FUNCTION_BLOCK FB_MoveSS_Exte
VAR_INPUT
	enable	:BOOL;
	ref		:AXIS_REF;
	jogF	:BOOL;
	jogB	:BOOL;
	Acceleration		:LREAL;
	Deceleration		:LREAL;
	Jerk				:LREAL;
END_VAR
VAR_OUTPUT	
END_VAR
VAR
	MC_Read:MC_ReadStatus;
	MC_ABS:MC_MoveAbsolute;
	MC_REL:MC_MoveRelative;
	MC_Jog:MC_Jog;
	
	MC_ABS1:MC_MoveAbsolute;
	MC_ABS2:MC_MoveAbsolute;
	MC_VELO:MC_MoveVelocity;
	
	step1,step2,step3		:INT;	
	R_TRIG1,R_TRIG2,R_TRIG3	:R_TRIG;
	R_TRIG_done				:R_TRIG;
	ton_NotMoving			:TON;
	ton_Moving				:TON;
	rel_do					:BOOL;
	abs_do					:BOOL;
	jogF_do					:BOOL;
	jogB_do					:BOOL;
	
	abs_do1,abs_do2,velo_do	:BOOL;
	error					:BOOL;

	MoveAbsolute_Busy		:BOOL;
	MoveConstantVelocity_Busy:BOOL;
	MoveRelative_Busy		:BOOL;
	jog_EN					:BOOL;
	FB_START_r_trig:		R_TRIG;
	start					:BOOL;
	jog_f_trig				:F_TRIG;
	ton_NotMoving_r_trig:Tc2_Standard.R_TRIG;
END_VAR
VAR_IN_OUT 
	MoveRelExe					:BOOL;
	MoveAbsExe					:BOOL;
	MoveConstantVelocityExe		:BOOL;//
	Velo						:LREAL;	//mm/s
	TargetRel					:LREAL;//mm
	TargetAbs					:LREAL;//mm
	constantvelocityStart		:LREAL;//mm		The position to start moving with a constant velocity
												//      0 < ConstantVelocityStart< ConstanVelocityEnd< RequestedPosition
	constanvelocityEnd			:LREAL;//mm		The position to end moving with a constant velocity											
	Done						:BOOL;
	NotMovingTimeOut 			:BOOL;
	SpeedNotReach				:BOOL;
END_VAR

(*********************NOT MOVING TIMEOUT***************************)
FB_START_r_trig(CLK:=jogF OR jogB OR MoveRelExe OR MoveAbsExe OR MoveConstantVelocityExe  , Q=> );
IF FB_START_r_trig.Q THEN 
	start:=TRUE;
END_IF
ton_NotMoving(IN:=Ref.Status.NotMoving AND start  , PT:= T#5S, Q=> , ET=> );
ton_NotMoving_r_trig(CLK:=ton_NotMoving.Q , Q=> );
IF ton_NotMoving_r_trig.Q THEN 
		NotMovingTimeOut:=TRUE;	
END_IF

Call_FB();
JOG();
MoveAbsolute();
MoveConstantVelocity();
MoveRelative();


(*********************error***************************)
IF ton_NotMoving.Q OR error OR SpeedNotReach THEN	
	start:=FALSE;
	error:=FALSE;
	ton_NotMoving(IN:=FALSE);	
	step1:=step2:=step2:=0;	
	MoveRelExe:=FALSE;
	MoveAbsExe:=FALSE;
	MoveConstantVelocityExe:=FALSE;
	Velo:=0;
	TargetAbs:=0;
	TargetRel:=0;
	constantvelocityStart:=0;
	constanvelocityend:=0;
	step1:=step2:=step3:=0;
	R_TRIG1(CLK:=FALSE);
	R_TRIG2(CLK:=FALSE);
	R_TRIG3(CLK:=FALSE);
END_IF

(*********************move done***************************)
IF MoveAbsolute_Busy OR MoveConstantVelocity_Busy OR  MoveRelative_Busy THEN 
	Done:=FALSE;
	jogF:=FALSE;
	jogB:=FALSE;
END_IF

jog_f_trig(CLK:=jogB OR jogF , Q=> );

R_TRIG_done(CLK:=MC_REL.Done OR MC_ABS.Done OR MC_ABS2.Done OR jog_f_trig.Q , Q=> );
IF R_TRIG_done.Q THEN 	
	start:=FALSE;
	R_TRIG_done(CLK:=FALSE);
	NotMovingTimeOut:=FALSE;
	ton_NotMoving(IN:=FALSE);
	step1:=step2:=step2:=0;	
	MoveRelExe:=FALSE;
	MoveAbsExe:=FALSE;
	MoveConstantVelocityExe:=FALSE;
	Velo:=0;
	TargetAbs:=0;
	TargetRel:=0;
	constantvelocityStart:=0;
	constanvelocityend:=0;
	Done:=TRUE ;
END_IF

ACTION Call_FB:
MC_Read(
	Axis:=ref , 
	Enable:=TRUE);
MC_REL(
	Axis:=ref , 
	Execute:=rel_do , 
	Distance:=TargetRel , 
	Velocity:=Velo , 
	Acceleration:=Acceleration , 
	Deceleration:=Deceleration , 
	Jerk:=Jerk , 
	BufferMode:= , 
	Options:= , 
	Done=> , 
	Busy=>MoveRelative_Busy , 
	Active=> , 
	CommandAborted=> , 
	Error=> , 
	ErrorID=> );
	IF MC_REL.Busy THEN 
		rel_do:=FALSE;
		MoveRelExe:=FALSE;
	END_IF
MC_ABS(
	Axis:=ref , 
	Execute:=abs_do , 
	Position:=TargetAbs , 
	Velocity:=Velo , 
	Acceleration:=Acceleration , 
	Deceleration:=Deceleration , 
	Jerk:=Jerk , 
	BufferMode:= , 
	Options:= , 
	Done=> , 
	Busy=>MoveAbsolute_Busy , 
	Active=> , 
	CommandAborted=> , 
	Error=> , 
	ErrorID=> );
	IF MC_ABS.Busy THEN 
		abs_do:=FALSE;
		MoveAbsExe:=FALSE;
	END_IF
MC_Jog(
	Axis:=ref , 
	JogForward:=jogF_do , 
	JogBackwards:=jogB_do , 
	Mode:=MC_JOGMODE_CONTINOUS , 
	Position:= , 
	Velocity:=Velo , 
	Acceleration:=Acceleration , 
	Deceleration:=Deceleration , 
	Jerk:=Jerk , 
	Done=> , 
	Busy=> , 
	Active=> , 
	CommandAborted=> , 
	Error=> , 
	ErrorID=> );
MC_ABS1(
	Axis:=ref , 
	Execute:=abs_do1 , 
	Position:=constanvelocityend , 
	Velocity:=Velo , 
	Acceleration:=Acceleration , 
	Deceleration:=Deceleration , 
	Jerk:=Jerk , 
	BufferMode:= , 
	Options:= , 
	Done=> , 
	Busy=> , 
	Active=> , 
	CommandAborted=> , 
	Error=> , 
	ErrorID=> );
	IF MC_ABS1.Busy THEN 
		abs_do1:=FALSE;
		MoveConstantVelocityExe:=FALSE;
	END_IF
MC_VELO(
	Axis:=ref , 
	Execute:=velo_do , 
	Velocity:=Velo , 
	Acceleration:=Acceleration , 
	Deceleration:=Deceleration , 
	Jerk:=Jerk , 
	Direction:= , 
	BufferMode:= MC_Aborting, 
	Options:= , 
	InVelocity=> , 
	Busy=> , 
	Active=> , 
	CommandAborted=> , 
	Error=> , 
	ErrorID=> );
	//IF MC_VELO.Busy THEN 
	//	velo_do:=FALSE;
	//END_IF
MC_ABS2(
	Axis:=ref , 
	Execute:=abs_do2 , 
	Position:=TargetAbs , 
	Velocity:=Velo , 
	Acceleration:=Acceleration , 
	Deceleration:=Deceleration , 
	Jerk:=Jerk , 
	BufferMode:=MC_Aborting , 
	Options:= , 
	Done=> , 
	Busy=> , 
	Active=> , 
	CommandAborted=> , 
	Error=> , 
	ErrorID=> );
	IF MC_ABS2.Busy THEN 
		abs_do2:=FALSE;
	END_IF
END_ACTION

ACTION JOG:
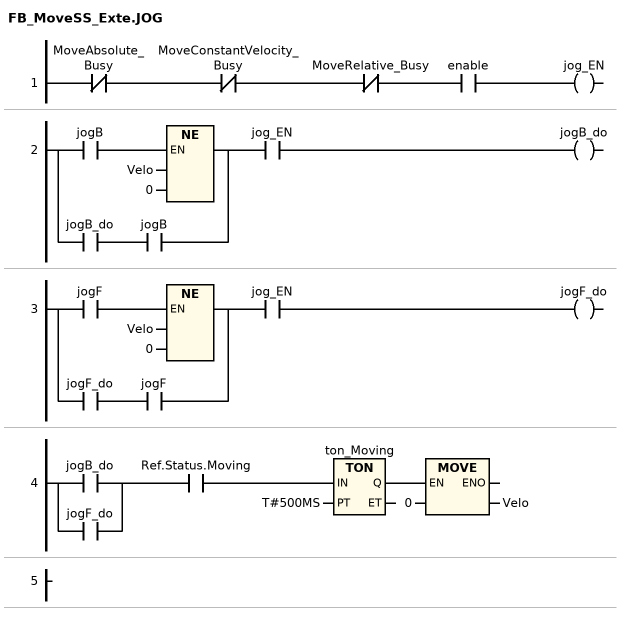
// NETWORK 1
jog_EN := NOT MoveAbsolute_Busy AND NOT MoveConstantVelocity_Busy AND NOT MoveRelative_Busy AND enable;

// NETWORK 2
jogB_do := (jogB AND Velo <> 0 OR jogB_do AND jogB) AND jog_EN;

// NETWORK 3
jogF_do := (jogF AND Velo <> 0 OR jogF_do AND jogF) AND jog_EN;

// NETWORK 4
ton_Moving(IN := (jogB_do OR jogF_do) AND Ref.Status.Moving, PT := T#500MS); // TON
IF ton_Moving.Q THEN Velo := 0; END_IF

// NETWORK 5
END_ACTION

ACTION MoveAbsolute:
(****************ABS********************)
R_TRIG2(CLK:=MoveAbsExe AND Ref.Status.NotMoving AND enable   , Q=> );

CASE step2 OF 
	0:				
		IF R_TRIG2.Q THEN 
			R_TRIG2(CLK:=FALSE);			
			MoveAbsExe:=FALSE;
			step2:=1;
		END_IF
	1:	
		IF   Velo<>0 THEN 		
			abs_do:=TRUE;
			step2:=2;
		END_IF
	2:
		IF MC_ABS.Busy THEN 
			abs_do:=FALSE;								
			step2 :=0;
		END_IF	
END_CASE


IF  MoveAbsolute_Busy THEN 
	MoveRelExe:=FALSE;
	MoveConstantVelocityExe:=FALSE;
END_IF
END_ACTION

ACTION MoveConstantVelocity:
(****************MoveConstantVelocity********************)
R_TRIG3(CLK:=MoveConstantVelocityExe AND Ref.Status.NotMoving AND enable  , Q=> );
CASE step3 OF 
	0:				
		IF R_TRIG3.Q THEN 
			R_TRIG3(CLK:=FALSE);
			MoveConstantVelocityExe:=FALSE;
			abs_do1:=abs_do2:=velo_do:=FALSE;		
			step3:=1;
		END_IF
	1:	//启动第一段，加速段
		IF   Velo<>0 THEN 		
			abs_do1:=TRUE;
			step3:=2;
		END_IF
		
	2:	//启动第二段，匀速段,增加到达位置时速度判断
		IF constanvelocityend>constantvelocityStart THEN 
			MC_VELO.Direction:=MC_Positive_Direction;
		ELSE
			MC_VELO.Direction:=MC_Negative_Direction;	
		END_IF
		
		IF 	(MC_VELO.Direction=MC_Positive_Direction AND ref.NcToPlc.ActPos>=constantvelocityStart)
			OR 	(MC_VELO.Direction=MC_Negative_Direction AND ref.NcToPlc.ActPos<=constantvelocityStart)  THEN 
			IF  ABS(ref.NcToPlc.ActVelo-velo)>10 THEN 
				abs_do1:=FALSE;	
				step3 :=5;
			END_IF
		END_IF
		
		IF ABS(ref.NcToPlc.ActVelo-velo)<=10 THEN			 
				abs_do1:=FALSE;					
				velo_do:=TRUE;									
				step3 :=3;
		END_IF
		
	3:	//启动第三段，减速段
		//IF MC_VELO.Busy THEN 
		//	velo_do:=FALSE;
		//END_IF
		IF (constanvelocityend>constantvelocityStart AND 
		 		ref.NcToPlc.ActPos>constanvelocityend)
		OR  (constanvelocityend<constantvelocityStart AND 
		 		ref.NcToPlc.ActPos<constanvelocityend)
		  THEN 	
			velo_do:=FALSE;
			abs_do2:=TRUE;
			step3 :=4;
		END_IF
	4:
		IF MC_ABS2.Busy THEN 
			abs_do2:=FALSE;
			step3 :=0;
		END_IF
	5://ERROR
		SpeedNotReach:=TRUE;
		step3 :=0;
		
END_CASE
MoveConstantVelocity_Busy:=MC_ABS1.Busy OR  MC_VELO.Busy OR MC_ABS2.Busy;

IF MoveConstantVelocity_Busy THEN 
	MoveRelExe:=FALSE;
	MoveAbsExe:=FALSE;
END_IF
END_ACTION

ACTION MoveConstantVelocity_old:
(****************MoveConstantVelocity********************)
R_TRIG3(CLK:=MoveConstantVelocityExe AND Ref.Status.NotMoving AND enable  , Q=> );
CASE step3 OF 
	0:				
		IF R_TRIG3.Q THEN 
			R_TRIG3(CLK:=FALSE);
			MoveConstantVelocityExe:=FALSE;
			abs_do1:=abs_do2:=velo_do:=FALSE;		
			step3:=1;
		END_IF
	1:	//启动第一段，加速段
		IF   Velo<>0 THEN 		
			abs_do1:=TRUE;
			step3:=2;
		END_IF
		
	2:	//启动第二段，匀速段,增加到达位置时速度判断
		IF constanvelocityend>constantvelocityStart THEN 
			MC_VELO.Direction:=MC_Positive_Direction;
		ELSE
			MC_VELO.Direction:=MC_Negative_Direction;	
		END_IF
		
		IF 	(MC_VELO.Direction=MC_Positive_Direction AND ref.NcToPlc.ActPos>=constantvelocityStart)
			OR 	(MC_VELO.Direction=MC_Negative_Direction AND ref.NcToPlc.ActPos<=constantvelocityStart)  THEN 
			IF NOT ref.Status.ConstantVelocity THEN 
				abs_do1:=FALSE;	
				step3 :=5;
			END_IF
		END_IF
		
		IF ref.Status.ConstantVelocity THEN			 
				abs_do1:=FALSE;					
				velo_do:=TRUE;									
				step3 :=3;
		END_IF
		
	3:	//启动第三段，减速段
		//IF MC_VELO.Busy THEN 
		//	velo_do:=FALSE;
		//END_IF
		IF (constanvelocityend>constantvelocityStart AND 
		 		ref.NcToPlc.ActPos>constanvelocityend)
		OR  (constanvelocityend<constantvelocityStart AND 
		 		ref.NcToPlc.ActPos<constanvelocityend)
		  THEN 	
			velo_do:=FALSE;
			abs_do2:=TRUE;
			step3 :=4;
		END_IF
	4:
		IF MC_ABS2.Busy THEN 
			abs_do2:=FALSE;
			step3 :=0;
		END_IF
	5://ERROR
		SpeedNotReach:=TRUE;
		step3 :=0;
		
END_CASE
MoveConstantVelocity_Busy:=MC_ABS1.Busy OR  MC_VELO.Busy OR MC_ABS2.Busy;

IF MoveConstantVelocity_Busy THEN 
	MoveRelExe:=FALSE;
	MoveAbsExe:=FALSE;
END_IF
END_ACTION

ACTION MoveRelative:
(****************Rel********************)
R_TRIG1(CLK:=MoveRelExe AND Ref.Status.NotMoving AND enable  , Q=> );
CASE step1 OF 
	0:				
		IF R_TRIG1.Q THEN 
			R_TRIG1(CLK:=FALSE);
			MoveRelExe:=FALSE;
			step1:=1;
		END_IF
	1:	
		IF TargetRel <>0 AND Velo<>0 THEN 		
			rel_do:=TRUE;
			step1:=2;
		END_IF
	2:
		IF MC_REL.Busy THEN 
			rel_do:=FALSE;								
			step1 :=0;
		END_IF	
END_CASE

IF MoveRelative_Busy THEN 
	MoveAbsExe:=FALSE;
	MoveConstantVelocityExe:=FALSE;
END_IF
END_ACTION

END_FUNCTION_BLOCK

(* stored: Version 1.1.0.1, ProductVersion 3.1.4024.11
   POU FB_MoveSS_Exte: Id {47959cd2-60f3-4e16-a2aa-8ba050a46cbb}, SpecialFunc None
   Action Call_FB: Id {bf29bd33-8141-4cc8-ab24-524dd322e163}
   Action JOG: Id {828fe6df-71e6-41bc-9e65-80a078ba92f1}
   Action MoveAbsolute: Id {79dfac2a-c87d-4714-a385-7c8b0a338777}
   Action MoveConstantVelocity: Id {6c76ece1-ec71-4593-9e1f-6680da88a89e}
   Action MoveConstantVelocity_old: Id {9ac806fc-5866-4cfe-a9da-ce0eb1deacac}
   Action MoveRelative: Id {27191e57-a8b2-4d22-b591-7f084cd3b093} *)
